Staubli VAL3: loadLibraries.pgx

program loadLibraries()
begin
//  nResult=scr:libLoad("Plastic/Modules/modScreen.zip","a81d706f651db0a6b2")
//  if nResult!=0
//    name=libPath()
//    nResult=scr:libLoad("Plastic/Modules/modScreen")
//    if nResult!=0
//      popUpMsg(name+":  Problem loading library for scr:")
//      call debug:error(libPath(),": Problem loading library for scr:")
//    else
//      call debug:info(libPath(),": Loading uncrypted version "+scr:libPath())
//    endIf
//  endIf
  // SECU
//  nResult=secu:libLoad("Plastic/Modules/modSafety.zip","a81d706f651db0a6b2")
//  if nResult!=0
//    name=libPath()
//    nResult=secu:libLoad("Plastic/Modules/modSafety")
//    if nResult!=0
//      popUpMsg(name+":  Problem loading library for secu:")
//      call debug:error(libPath(),": Problem loading library for secu:")
//    else
//      call debug:info(libPath(),": Loading uncrypted version "+secu:libPath())
//    endIf
//  endIf
//  // STATUS
//  nResult=stat:libLoad("Plastic/Modules/modStatus.zip","a81d706f651db0a6b2")
//  if nResult!=0
//    name=libPath()
//    nResult=stat:libLoad("Plastic/Modules/modStatus")
//    if nResult!=0
//      popUpMsg(name+":  Problem loading library for stat:")
//      call debug:error(libPath(),": Problem loading library for stat:")
//    else
//      call debug:info(libPath(),": Loading uncrypted version "+stat:libPath())
//    endIf
//  endIf
end
